// Writes a fixed32 field value, without a tag, to the stream.
FUNCTION F_WriteFixed32 : HRESULT
VAR_IN_OUT
    aBuffer : ARRAY [*] OF BYTE;
    stState : ST_WriterInternalState;
END_VAR
VAR_INPUT
    nValue : UDINT;
END_VAR
VAR
END_VAR

F_WriteFixed32 := F_WriteRawLittleEndian32(aBuffer, stState, nValue);

END_FUNCTION

(* stored: Version 1.1.0.1
   POU F_WriteFixed32: Id {1c0274d5-4789-43a4-9ff5-fd680c0bf1d5}, SpecialFunc None *)
